LIN {X 0,Y 83.4,Z 651.34,A -85,B 0,C 180,E1 -27838.974,E2 -27838.974} C_VEL
LIN {X 0,Y 87.355,Z 640.881,A -85,B 0,C 180,E1 -27845.629,E2 -27845.629} C_VEL
LIN {X 0,Y 92.332,Z 628.192,A -85,B 0,C 180,E1 -27851.751,E2 -27851.751} C_VEL
LIN {X 0,Y 97.709,Z 614.337,A -85,B 0,C 180,E1 -27856.732,E2 -27856.732} C_VEL
LIN {X 0,Y 102.843,Z 599.666,A -85,B 0,C 180,E1 -27860.677,E2 -27860.677} C_VEL
LIN {X 0,Y 107.389,Z 585.24,A -85,B 0,C 180,E1 -27863.541,E2 -27863.541} C_VEL
LIN {X 0,Y 110.995,Z 571.561,A -85,B 0,C 180,E1 -27865.587,E2 -27865.587} C_VEL
LIN {X 0,Y 111.796,Z 565.957,A -85,B 0,C 180,E1 -27866.44,E2 -27866.44} C_VEL
LIN {X 0,Y 111.242,Z 556.652,A -85,B 0,C 180,E1 -27868.182,E2 -27868.182} C_VEL
LIN {X 0,Y 110.441,Z 547.232,A -85,B 0,C 180,E1 -27869.834,E2 -27869.834} C_VEL
LIN {X 0,Y 110.751,Z 541.433,A -85,B 0,C 180,E1 -27870.482,E2 -27870.482} C_VEL
LIN {X 0,Y 118.536,Z 490.469,A -85,B 0,C 180,E1 -27874.19,E2 -27874.19} C_VEL
LIN {X 0,Y 112.616,Z 471.763,A -85,B 0,C 180,E1 -27879.39,E2 -27879.39} C_VEL
LIN {X 0,Y 109.271,Z 463.872,A -85,B 0,C 180,E1 -27882.247,E2 -27882.247} C_VEL
LIN {X 0,Y 104.426,Z 453.54,A -85,B 0,C 180,E1 -27886.806,E2 -27886.806} C_VEL
LIN {X 0,Y 99.664,Z 444.282,A -85,B 0,C 180,E1 -27891.893,E2 -27891.893} C_VEL
LIN {X 0,Y 95.134,Z 435.831,A -85,B 0,C 180,E1 -27897.713,E2 -27897.713} C_VEL
LIN {X 0,Y 91.912,Z 430.585,A -85,B 0,C 180,E1 -27902.471,E2 -27902.471} C_VEL
LIN {X 0,Y 90.145,Z 427.655,A -85,B 0,C 180,E1 -27905.52,E2 -27905.52} C_VEL
LIN {X 0,Y 87.765,Z 424.651,A -85,B 0,C 180,E1 -27910.178,E2 -27910.178} C_VEL
LIN {X 0,Y 87.158,Z 423.342,A -85,B 0,C 180,E1 -27911.706,E2 -27911.706} C_VEL
LIN {X 0,Y 83.913,Z 420.372,A -85,B 0,C 180,E1 -27920.293,E2 -27920.293} C_VEL
LIN {X 0,Y 83.066,Z 418.058,A -85,B 0,C 180,E1 -27925.028,E2 -27925.028} C_VEL
LIN {X 0,Y 81.987,Z 417.702,A -85,B 0,C 180,E1 -27939.525,E2 -27939.525} C_VEL
LIN {X 0,Y 82.984,Z 418.172,A -85,B 0,C 180,E1 -27946.706,E2 -27946.706} C_VEL
LIN {X 0,Y 84.247,Z 421.149,A -85,B 0,C 180,E1 -27953.039,E2 -27953.039} C_VEL
LIN {X 0,Y 86.921,Z 423.772,A -85,B 0,C 180,E1 -27959.99,E2 -27959.99} C_VEL
LIN {X 0,Y 88.86,Z 427.056,A -85,B 0,C 180,E1 -27964.348,E2 -27964.348} C_VEL
LIN {X 0,Y 90.285,Z 428.713,A -85,B 0,C 180,E1 -27966.89,E2 -27966.89} C_VEL
LIN {X 0,Y 92.73,Z 432.159,A -85,B 0,C 180,E1 -27970.786,E2 -27970.786} C_VEL
LIN {X 0,Y 96.209,Z 437.6,A -85,B 0,C 180,E1 -27975.639,E2 -27975.639} C_VEL
LIN {X 0,Y 99.737,Z 443.153,A -85,B 0,C 180,E1 -27979.836,E2 -27979.836} C_VEL
LIN {X 0,Y 105.389,Z 454.817,A -85,B 0,C 180,E1 -27985.913,E2 -27985.913} C_VEL
LIN {X 0,Y 111.16,Z 468.054,A -85,B 0,C 180,E1 -27991.255,E2 -27991.255} C_VEL
LIN {X 0,Y 116.833,Z 481.707,A -85,B 0,C 180,E1 -27995.829,E2 -27995.829} C_VEL
LIN {X 0,Y 118.524,Z 486.01,A -85,B 0,C 180,E1 -27997.101,E2 -27997.101} C_VEL
LIN {X 0,Y 108.606,Z 548.727,A -85,B 0,C 180,E1 -28001.636,E2 -28001.636} C_VEL
LIN {X 0,Y 105.23,Z 564.977,A -85,B 0,C 180,E1 -28003.441,E2 -28003.441} C_VEL
LIN {X 0,Y 100.84,Z 581.24,A -85,B 0,C 180,E1 -28005.969,E2 -28005.969} C_VEL
LIN {X 0,Y 95.78,Z 596.719,A -85,B 0,C 180,E1 -28009.296,E2 -28009.296} C_VEL
LIN {X 0,Y 90.179,Z 611.69,A -85,B 0,C 180,E1 -28013.687,E2 -28013.687} C_VEL
LIN {X 0,Y 84.987,Z 624.642,A -85,B 0,C 180,E1 -28018.821,E2 -28018.821} C_VEL
LIN {X 0,Y 79.8,Z 637.202,A -85,B 0,C 180,E1 -28025.445,E2 -28025.445} C_VEL
LIN {X 0,Y 75.323,Z 648.898,A -85,B 0,C 180,E1 -28033.686,E2 -28033.686} C_VEL
LIN {X 0,Y 72.406,Z 658.262,A -85,B 0,C 180,E1 -28042.329,E2 -28042.329} C_VEL
LIN {X 0,Y 70.888,Z 665.175,A -85,B 0,C 180,E1 -28050.282,E2 -28050.282} C_VEL
LIN {X 0,Y 70.041,Z 671.752,A -85,B 0,C 180,E1 -28059.438,E2 -28059.438} C_VEL
LIN {X 0,Y 70.296,Z 677.109,A -85,B 0,C 180,E1 -28068.464,E2 -28068.464} C_VEL
LIN {X 0,Y 72.587,Z 682.826,A -85,B 0,C 180,E1 -28079.998,E2 -28079.998} C_VEL
LIN {X 0,Y 77.201,Z 687.278,A -85,B 0,C 180,E1 -28090.489,E2 -28090.489} C_VEL
LIN {X 0,Y 84.118,Z 690.712,A -85,B 0,C 180,E1 -28099.522,E2 -28099.522} C_VEL
LIN {X 0,Y 92.853,Z 693.253,A -85,B 0,C 180,E1 -28107.008,E2 -28107.008} C_VEL
LIN {X 0,Y 104.49,Z 695.039,A -85,B 0,C 180,E1 -28113.751,E2 -28113.751} C_VEL
LIN {X 0,Y 103.442,Z 695.069,A -85,B 0,C 180,E1 -28115.374,E2 -28115.374} C_VEL
LIN {X 0,Y 93.415,Z 694.243,A -85,B 0,C 180,E1 -28121.198,E2 -28121.198} C_VEL
LIN {X 0,Y 84.648,Z 692.545,A -85,B 0,C 180,E1 -28128.37,E2 -28128.37} C_VEL
LIN {X 0,Y 77.842,Z 690.142,A -85,B 0,C 180,E1 -28137.191,E2 -28137.191} C_VEL
LIN {X 0,Y 72.686,Z 685.827,A -85,B 0,C 180,E1 -28150.211,E2 -28150.211} C_VEL
LIN {X 0,Y 71.425,Z 680.817,A -85,B 0,C 180,E1 -28162.373,E2 -28162.373} C_VEL
LIN {X 0,Y 71.518,Z 678.411,A -85,B 0,C 180,E1 -28167.175,E2 -28167.175} C_VEL
LIN {X 0,Y 71.275,Z 673.088,A -85,B 0,C 180,E1 -28175.65,E2 -28175.65} C_VEL
LIN {X 0,Y 72.103,Z 665.419,A -85,B 0,C 180,E1 -28185.539,E2 -28185.539} C_VEL
LIN {X 0,Y 74.517,Z 655.967,A -85,B 0,C 180,E1 -28195.104,E2 -28195.104} C_VEL
LIN {X 0,Y 78.723,Z 644.592,A -85,B 0,C 180,E1 -28203.906,E2 -28203.906} C_VEL
LIN {X 0,Y 83.249,Z 633.196,A -85,B 0,C 180,E1 -28210.556,E2 -28210.556} C_VEL
LIN {X 0,Y 88.734,Z 620.083,A -85,B 0,C 180,E1 -28216.27,E2 -28216.27} C_VEL
LIN {X 0,Y 93.537,Z 607.632,A -85,B 0,C 180,E1 -28220.356,E2 -28220.356} C_VEL
LIN {X 0,Y 98.821,Z 592.668,A -85,B 0,C 180,E1 -28223.984,E2 -28223.984} C_VEL
LIN {X 0,Y 103.223,Z 577.827,A -85,B 0,C 180,E1 -28226.649,E2 -28226.649} C_VEL
LIN {X 0,Y 106.858,Z 562.938,A -85,B 0,C 180,E1 -28228.602,E2 -28228.602} C_VEL
LIN {X 0,Y 109.639,Z 548.688,A -85,B 0,C 180,E1 -28229.913,E2 -28229.913} C_VEL
LIN {X 0,Y 110.751,Z 541.433,A -85,B 0,C 180,E1 -28230.482,E2 -28230.482} C_VEL
LIN {X 0,Y 111.09,Z 535.664,A -85,B 0,C 180,E1 -28231.12,E2 -28231.12} C_VEL
LIN {X 0,Y 109.501,Z 516.872,A -85,B 0,C 180,E1 -28234.326,E2 -28234.326} C_VEL
LIN {X 0,Y 109.908,Z 511.103,A -85,B 0,C 180,E1 -28234.962,E2 -28234.962} C_VEL
LIN {X 0,Y 112.849,Z 492.252,A -85,B 0,C 180,E1 -28236.331,E2 -28236.331} C_VEL
LIN {X 0,Y 107.793,Z 475.639,A -85,B 0,C 180,E1 -28241.188,E2 -28241.188} C_VEL
LIN {X 0,Y 104.92,Z 468.523,A -85,B 0,C 180,E1 -28243.921,E2 -28243.921} C_VEL
LIN {X 0,Y 100.246,Z 458.053,A -85,B 0,C 180,E1 -28248.824,E2 -28248.824} C_VEL
LIN {X 0,Y 95.193,Z 447.833,A -85,B 0,C 180,E1 -28254.835,E2 -28254.835} C_VEL
LIN {X 0,Y 91.737,Z 441.143,A -85,B 0,C 180,E1 -28259.869,E2 -28259.869} C_VEL
LIN {X 0,Y 89.106,Z 436.502,A -85,B 0,C 180,E1 -28264.187,E2 -28264.187} C_VEL
LIN {X 0,Y 87.569,Z 433.904,A -85,B 0,C 180,E1 -28267.147,E2 -28267.147} C_VEL
LIN {X 0,Y 85.254,Z 430.535,A -85,B 0,C 180,E1 -28272.22,E2 -28272.22} C_VEL
LIN {X 0,Y 84.709,Z 429.774,A -85,B 0,C 180,E1 -28273.543,E2 -28273.543} C_VEL
LIN {X 0,Y 82.042,Z 426.845,A -85,B 0,C 180,E1 -28281.915,E2 -28281.915} C_VEL
LIN {X 0,Y 81.443,Z 425.088,A -85,B 0,C 180,E1 -28285.562,E2 -28285.562} C_VEL
LIN {X 0,Y 80.477,Z 424.626,A -85,B 0,C 180,E1 -28298.203,E2 -28298.203} C_VEL
LIN {X 0,Y 81.333,Z 425.135,A -85,B 0,C 180,E1 -28305.96,E2 -28305.96} C_VEL
LIN {X 0,Y 83.041,Z 428.687,A -85,B 0,C 180,E1 -28314.159,E2 -28314.159} C_VEL
LIN {X 0,Y 84.78,Z 430.442,A -85,B 0,C 180,E1 -28318.804,E2 -28318.804} C_VEL
LIN {X 0,Y 86.896,Z 433.84,A -85,B 0,C 180,E1 -28323.684,E2 -28323.684} C_VEL
LIN {X 0,Y 87.932,Z 435.321,A -85,B 0,C 180,E1 -28325.758,E2 -28325.758} C_VEL
LIN {X 0,Y 90.71,Z 439.474,A -85,B 0,C 180,E1 -28330.503,E2 -28330.503} C_VEL
LIN {X 0,Y 93.875,Z 444.671,A -85,B 0,C 180,E1 -28335.078,E2 -28335.078} C_VEL
LIN {X 0,Y 96.373,Z 448.911,A -85,B 0,C 180,E1 -28338.317,E2 -28338.317} C_VEL
LIN {X 0,Y 101.476,Z 460.012,A -85,B 0,C 180,E1 -28344.265,E2 -28344.265} C_VEL
LIN {X 0,Y 106.79,Z 472.868,A -85,B 0,C 180,E1 -28349.725,E2 -28349.725} C_VEL
LIN {X 0,Y 112.767,Z 487.766,A -85,B 0,C 180,E1 -28354.863,E2 -28354.863} C_VEL
LIN {X 0,Y 104.427,Z 539.915,A -85,B 0,C 180,E1 -28358.697,E2 -28358.697} C_VEL
LIN {X 0,Y 101.113,Z 557.125,A -85,B 0,C 180,E1 -28360.273,E2 -28360.273} C_VEL
LIN {X 0,Y 97.417,Z 572.043,A -85,B 0,C 180,E1 -28362.273,E2 -28362.273} C_VEL
LIN {X 0,Y 92.422,Z 588.129,A -85,B 0,C 180,E1 -28365.244,E2 -28365.244} C_VEL
LIN {X 0,Y 86.759,Z 603.763,A -85,B 0,C 180,E1 -28369.273,E2 -28369.273} C_VEL
LIN {X 0,Y 80.958,Z 617.943,A -85,B 0,C 180,E1 -28374.287,E2 -28374.287} C_VEL
LIN {X 0,Y 75.457,Z 630.788,A -85,B 0,C 180,E1 -28380.507,E2 -28380.507} C_VEL
LIN {X 0,Y 70.887,Z 641.562,A -85,B 0,C 180,E1 -28387.517,E2 -28387.517} C_VEL
LIN {X 0,Y 67.145,Z 651.543,A -85,B 0,C 180,E1 -28396.049,E2 -28396.049} C_VEL
LIN {X 0,Y 64.435,Z 661.363,A -85,B 0,C 180,E1 -28406.949,E2 -28406.949} C_VEL
LIN {X 0,Y 63.243,Z 668.627,A -85,B 0,C 180,E1 -28417.109,E2 -28417.109} C_VEL
LIN {X 0,Y 63.267,Z 674.398,A -85,B 0,C 180,E1 -28427.162,E2 -28427.162} C_VEL
LIN {X 0,Y 65.417,Z 680.637,A -85,B 0,C 180,E1 -28439.998,E2 -28439.998} C_VEL
LIN {X 0,Y 70.149,Z 685.571,A -85,B 0,C 180,E1 -28451.557,E2 -28451.557} C_VEL
LIN {X 0,Y 77.355,Z 689.428,A -85,B 0,C 180,E1 -28461.309,E2 -28461.309} C_VEL
LIN {X 0,Y 86.428,Z 692.389,A -85,B 0,C 180,E1 -28469.201,E2 -28469.201} C_VEL
LIN {X 0,Y 91.847,Z 693.586,A -85,B 0,C 180,E1 -28472.668,E2 -28472.668} C_VEL
LIN {X 0,Y 94.095,Z 694.045,A -85,B 0,C 180,E1 -28474.745,E2 -28474.745} C_VEL
LIN {X 0,Y 79.518,Z 691.492,A -85,B 0,C 180,E1 -28484.994,E2 -28484.994} C_VEL
LIN {X 0,Y 69.224,Z 687.122,A -85,B 0,C 180,E1 -28499.485,E2 -28499.485} C_VEL
LIN {X 0,Y 65.545,Z 683.066,A -85,B 0,C 180,E1 -28511.226,E2 -28511.226} C_VEL
LIN {X 0,Y 64.721,Z 677.982,A -85,B 0,C 180,E1 -28523.757,E2 -28523.757} C_VEL
LIN {X 0,Y 64.541,Z 674.68,A -85,B 0,C 180,E1 -28529.991,E2 -28529.991} C_VEL
LIN {X 0,Y 64.449,Z 669.034,A -85,B 0,C 180,E1 -28538.816,E2 -28538.816} C_VEL
LIN {X 0,Y 65.361,Z 662.721,A -85,B 0,C 180,E1 -28547.19,E2 -28547.19} C_VEL
LIN {X 0,Y 68.239,Z 652.923,A -85,B 0,C 180,E1 -28557.6,E2 -28557.6} C_VEL
LIN {X 0,Y 72.206,Z 642.852,A -85,B 0,C 180,E1 -28565.721,E2 -28565.721} C_VEL
LIN {X 0,Y 77.472,Z 630.305,A -85,B 0,C 180,E1 -28573.246,E2 -28573.246} C_VEL
LIN {X 0,Y 82.941,Z 617.719,A -85,B 0,C 180,E1 -28578.754,E2 -28578.754} C_VEL
LIN {X 0,Y 88.624,Z 603.293,A -85,B 0,C 180,E1 -28583.398,E2 -28583.398} C_VEL
LIN {X 0,Y 94.231,Z 587.487,A -85,B 0,C 180,E1 -28587.028,E2 -28587.028} C_VEL
LIN {X 0,Y 99.038,Z 570.951,A -85,B 0,C 180,E1 -28589.755,E2 -28589.755} C_VEL
LIN {X 0,Y 102.85,Z 554.608,A -85,B 0,C 180,E1 -28591.605,E2 -28591.605} C_VEL
LIN {X 0,Y 109.908,Z 511.103,A -85,B 0,C 180,E1 -28594.962,E2 -28594.962} C_VEL
LIN {X 0,Y 110.223,Z 507.254,A -85,B 0,C 180,E1 -28595.373,E2 -28595.373} C_VEL
LIN {X 0,Y 109.773,Z 501.658,A -85,B 0,C 180,E1 -28596.38,E2 -28596.38} C_VEL
LIN {X 0,Y 108.55,Z 496.379,A -85,B 0,C 180,E1 -28597.708,E2 -28597.708} C_VEL
LIN {X 0,Y 104.028,Z 482.75,A -85,B 0,C 180,E1 -28602.073,E2 -28602.073} C_VEL
LIN {X 0,Y 101.897,Z 476.229,A -85,B 0,C 180,E1 -28604.416,E2 -28604.416} C_VEL
LIN {X 0,Y 97.693,Z 466.124,A -85,B 0,C 180,E1 -28609.06,E2 -28609.06} C_VEL
LIN {X 0,Y 93.087,Z 455.985,A -85,B 0,C 180,E1 -28614.877,E2 -28614.877} C_VEL
LIN {X 0,Y 88.893,Z 447.211,A -85,B 0,C 180,E1 -28621.353,E2 -28621.353} C_VEL
LIN {X 0,Y 85.396,Z 440.486,A -85,B 0,C 180,E1 -28628.172,E2 -28628.172} C_VEL
LIN {X 0,Y 82.991,Z 436.835,A -85,B 0,C 180,E1 -28633.829,E2 -28633.829} C_VEL
LIN {X 0,Y 80.039,Z 432.914,A -85,B 0,C 180,E1 -28644.512,E2 -28644.512} C_VEL
LIN {X 0,Y 79.66,Z 431.821,A -85,B 0,C 180,E1 -28647.249,E2 -28647.249} C_VEL
LIN {X 0,Y 79.032,Z 431.568,A -85,B 0,C 180,E1 -28658.499,E2 -28658.499} C_VEL
LIN {X 0,Y 79.693,Z 432.069,A -85,B 0,C 180,E1 -28665.141,E2 -28665.141} C_VEL
LIN {X 0,Y 81.687,Z 435.942,A -85,B 0,C 180,E1 -28674.737,E2 -28674.737} C_VEL
LIN {X 0,Y 82.616,Z 436.923,A -85,B 0,C 180,E1 -28677.368,E2 -28677.368} C_VEL
LIN {X 0,Y 84.684,Z 440.337,A -85,B 0,C 180,E1 -28682.492,E2 -28682.492} C_VEL
LIN {X 0,Y 87.851,Z 445.4,A -85,B 0,C 180,E1 -28688.793,E2 -28688.793} C_VEL
LIN {X 0,Y 91.961,Z 452.355,A -85,B 0,C 180,E1 -28695.059,E2 -28695.059} C_VEL
LIN {X 0,Y 95.16,Z 459.605,A -85,B 0,C 180,E1 -28699.602,E2 -28699.602} C_VEL
LIN {X 0,Y 98.909,Z 468.618,A -85,B 0,C 180,E1 -28704.153,E2 -28704.153} C_VEL
LIN {X 0,Y 103.142,Z 479.356,A -85,B 0,C 180,E1 -28708.74,E2 -28708.74} C_VEL
LIN {X 0,Y 107.174,Z 489.956,A -85,B 0,C 180,E1 -28712.58,E2 -28712.58} C_VEL
LIN {X 0,Y 97.537,Z 546.504,A -85,B 0,C 180,E1 -28716.792,E2 -28716.792} C_VEL
LIN {X 0,Y 93.909,Z 563.2,A -85,B 0,C 180,E1 -28718.615,E2 -28718.615} C_VEL
LIN {X 0,Y 89.493,Z 578.67,A -85,B 0,C 180,E1 -28720.988,E2 -28720.988} C_VEL
LIN {X 0,Y 84.193,Z 594.018,A -85,B 0,C 180,E1 -28724.27,E2 -28724.27} C_VEL
LIN {X 0,Y 78.687,Z 607.907,A -85,B 0,C 180,E1 -28728.375,E2 -28728.375} C_VEL
LIN {X 0,Y 72.79,Z 621.401,A -85,B 0,C 180,E1 -28733.928,E2 -28733.928} C_VEL
LIN {X 0,Y 67.266,Z 633.472,A -85,B 0,C 180,E1 -28740.755,E2 -28740.755} C_VEL
LIN {X 0,Y 62.856,Z 643.63,A -85,B 0,C 180,E1 -28748.491,E2 -28748.491} C_VEL
LIN {X 0,Y 58.974,Z 654.059,A -85,B 0,C 180,E1 -28759.045,E2 -28759.045} C_VEL
LIN {X 0,Y 57.067,Z 662.089,A -85,B 0,C 180,E1 -28769.57,E2 -28769.57} C_VEL
LIN {X 0,Y 56.252,Z 668.459,A -85,B 0,C 180,E1 -28779.903,E2 -28779.903} C_VEL
LIN {X 0,Y 56.928,Z 675.031,A -85,B 0,C 180,E1 -28792.906,E2 -28792.906} C_VEL
LIN {X 0,Y 60.395,Z 681.051,A -85,B 0,C 180,E1 -28806.681,E2 -28806.681} C_VEL
LIN {X 0,Y 66.738,Z 685.963,A -85,B 0,C 180,E1 -28818.575,E2 -28818.575} C_VEL
LIN {X 0,Y 80.183,Z 691.258,A -85,B 0,C 180,E1 -28831.727,E2 -28831.727} C_VEL
LIN {X 0,Y 83.422,Z 692.126,A -85,B 0,C 180,E1 -28833.87,E2 -28833.87} C_VEL
LIN {X 0,Y 82.706,Z 692.041,A -85,B 0,C 180,E1 -28835.271,E2 -28835.271} C_VEL
LIN {X 0,Y 70.348,Z 688.871,A -85,B 0,C 180,E1 -28845.616,E2 -28845.616} C_VEL
LIN {X 0,Y 61.987,Z 684.558,A -85,B 0,C 180,E1 -28859.312,E2 -28859.312} C_VEL
LIN {X 0,Y 58.146,Z 678.749,A -85,B 0,C 180,E1 -28876.001,E2 -28876.001} C_VEL
LIN {X 0,Y 57.98,Z 675.904,A -85,B 0,C 180,E1 -28883.027,E2 -28883.027} C_VEL
LIN {X 0,Y 57.654,Z 672.44,A -85,B 0,C 180,E1 -28889.99,E2 -28889.99} C_VEL
LIN {X 0,Y 57.853,Z 664.848,A -85,B 0,C 180,E1 -28902.383,E2 -28902.383} C_VEL
LIN {X 0,Y 59.921,Z 655.642,A -85,B 0,C 180,E1 -28914.226,E2 -28914.226} C_VEL
LIN {X 0,Y 63.499,Z 646.207,A -85,B 0,C 180,E1 -28923.589,E2 -28923.589} C_VEL
LIN {X 0,Y 68.404,Z 635.031,A -85,B 0,C 180,E1 -28931.887,E2 -28931.887} C_VEL
LIN {X 0,Y 74.016,Z 622.74,A -85,B 0,C 180,E1 -28938.507,E2 -28938.507} C_VEL
LIN {X 0,Y 79.672,Z 609.635,A -85,B 0,C 180,E1 -28943.59,E2 -28943.59} C_VEL
LIN {X 0,Y 85.281,Z 595.268,A -85,B 0,C 180,E1 -28947.625,E2 -28947.625} C_VEL
LIN {X 0,Y 90.263,Z 580.691,A -85,B 0,C 180,E1 -28950.569,E2 -28950.569} C_VEL
LIN {X 0,Y 94.704,Z 564.576,A -85,B 0,C 180,E1 -28952.924,E2 -28952.924} C_VEL
LIN {X 0,Y 98.01,Z 549.43,A -85,B 0,C 180,E1 -28954.432,E2 -28954.432} C_VEL
LIN {X 0,Y 107.266,Z 493.905,A -85,B 0,C 180,E1 -28958.669,E2 -28958.669} C_VEL
LIN {X 0,Y 104.028,Z 482.75,A -85,B 0,C 180,E1 -28962.073,E2 -28962.073} C_VEL
LIN {X 0,Y 102.842,Z 479.687,A -85,B 0,C 180,E1 -28963.257,E2 -28963.257} C_VEL
LIN {X 0,Y 101.281,Z 477.066,A -85,B 0,C 180,E1 -28964.65,E2 -28964.65} C_VEL
LIN {X 0,Y 97.595,Z 472.757,A -85,B 0,C 180,E1 -28967.863,E2 -28967.863} C_VEL
LIN {X 0,Y 92.154,Z 466.593,A -85,B 0,C 180,E1 -28973.301,E2 -28973.301} C_VEL
LIN {X 0,Y 90.821,Z 464.06,A -85,B 0,C 180,E1 -28975.089,E2 -28975.089} C_VEL
LIN {X 0,Y 87.082,Z 455.522,A -85,B 0,C 180,E1 -28981.123,E2 -28981.123} C_VEL
LIN {X 0,Y 84.081,Z 449.056,A -85,B 0,C 180,E1 -28987.141,E2 -28987.141} C_VEL
LIN {X 0,Y 82.634,Z 446.346,A -85,B 0,C 180,E1 -28990.546,E2 -28990.546} C_VEL
LIN {X 0,Y 80.518,Z 442.925,A -85,B 0,C 180,E1 -28996.261,E2 -28996.261} C_VEL
LIN {X 0,Y 78.408,Z 439.849,A -85,B 0,C 180,E1 -29005.056,E2 -29005.056} C_VEL
LIN {X 0,Y 78.132,Z 438.722,A -85,B 0,C 180,E1 -29007.544,E2 -29007.544} C_VEL
LIN {X 0,Y 77.592,Z 438.548,A -85,B 0,C 180,E1 -29019.35,E2 -29019.35} C_VEL
LIN {X 0,Y 78.054,Z 438.9,A -85,B 0,C 180,E1 -29024.166,E2 -29024.166} C_VEL
LIN {X 0,Y 80,Z 442.817,A -85,B 0,C 180,E1 -29034.273,E2 -29034.273} C_VEL
LIN {X 0,Y 80.584,Z 443.656,A -85,B 0,C 180,E1 -29036.173,E2 -29036.173} C_VEL
LIN {X 0,Y 83.15,Z 448.015,A -85,B 0,C 180,E1 -29042.862,E2 -29042.862} C_VEL
LIN {X 0,Y 85.387,Z 452.007,A -85,B 0,C 180,E1 -29047.626,E2 -29047.626} C_VEL
LIN {X 0,Y 89.135,Z 458.751,A -85,B 0,C 180,E1 -29053.85,E2 -29053.85} C_VEL
LIN {X 0,Y 93.266,Z 469.238,A -85,B 0,C 180,E1 -29060.117,E2 -29060.117} C_VEL
LIN {X 0,Y 97.709,Z 481.044,A -85,B 0,C 180,E1 -29065.657,E2 -29065.657} C_VEL
LIN {X 0,Y 101.664,Z 491.965,A -85,B 0,C 180,E1 -29070.006,E2 -29070.006} C_VEL
LIN {X 0,Y 92.249,Z 545.502,A -85,B 0,C 180,E1 -29073.99,E2 -29073.99} C_VEL
LIN {X 0,Y 88.314,Z 563.044,A -85,B 0,C 180,E1 -29075.865,E2 -29075.865} C_VEL
LIN {X 0,Y 83.737,Z 578.397,A -85,B 0,C 180,E1 -29078.236,E2 -29078.236} C_VEL
LIN {X 0,Y 78.051,Z 594.121,A -85,B 0,C 180,E1 -29081.692,E2 -29081.692} C_VEL
LIN {X 0,Y 72.056,Z 608.35,A -85,B 0,C 180,E1 -29086.115,E2 -29086.115} C_VEL
LIN {X 0,Y 65.548,Z 622.429,A -85,B 0,C 180,E1 -29092.362,E2 -29092.362} C_VEL
LIN {X 0,Y 60.129,Z 633.728,A -85,B 0,C 180,E1 -29099.376,E2 -29099.376} C_VEL
LIN {X 0,Y 55.616,Z 643.71,A -85,B 0,C 180,E1 -29107.83,E2 -29107.83} C_VEL
LIN {X 0,Y 51.683,Z 654.011,A -85,B 0,C 180,E1 -29119.762,E2 -29119.762} C_VEL
LIN {X 0,Y 49.98,Z 661.315,A -85,B 0,C 180,E1 -29130.728,E2 -29130.728} C_VEL
LIN {X 0,Y 49.357,Z 668.196,A -85,B 0,C 180,E1 -29143.452,E2 -29143.452} C_VEL
LIN {X 0,Y 50.449,Z 673.878,A -85,B 0,C 180,E1 -29156.004,E2 -29156.004} C_VEL
LIN {X 0,Y 54.731,Z 680.068,A -85,B 0,C 180,E1 -29171.103,E2 -29171.103} C_VEL
LIN {X 0,Y 64.175,Z 686.139,A -85,B 0,C 180,E1 -29185.978,E2 -29185.978} C_VEL
LIN {X 0,Y 72.799,Z 689.489,A -85,B 0,C 180,E1 -29193.716,E2 -29193.716} C_VEL
LIN {X 0,Y 70.312,Z 688.905,A -85,B 0,C 180,E1 -29196.891,E2 -29196.891} C_VEL
LIN {X 0,Y 57.716,Z 683.811,A -85,B 0,C 180,E1 -29212.482,E2 -29212.482} C_VEL
LIN {X 0,Y 52.746,Z 679.298,A -85,B 0,C 180,E1 -29226.427,E2 -29226.427} C_VEL
LIN {X 0,Y 51.285,Z 673.685,A -85,B 0,C 180,E1 -29242.112,E2 -29242.112} C_VEL
LIN {X 0,Y 50.807,Z 670.005,A -85,B 0,C 180,E1 -29249.988,E2 -29249.988} C_VEL
LIN {X 0,Y 51.013,Z 662.528,A -85,B 0,C 180,E1 -29263.361,E2 -29263.361} C_VEL
LIN {X 0,Y 53.66,Z 652.473,A -85,B 0,C 180,E1 -29277.271,E2 -29277.271} C_VEL
LIN {X 0,Y 57.809,Z 642.526,A -85,B 0,C 180,E1 -29287.421,E2 -29287.421} C_VEL
LIN {X 0,Y 62.827,Z 631.726,A -85,B 0,C 180,E1 -29295.476,E2 -29295.476} C_VEL
LIN {X 0,Y 69.339,Z 618.186,A -85,B 0,C 180,E1 -29302.62,E2 -29302.62} C_VEL
LIN {X 0,Y 75.063,Z 605.299,A -85,B 0,C 180,E1 -29307.405,E2 -29307.405} C_VEL
LIN {X 0,Y 81.086,Z 590.294,A -85,B 0,C 180,E1 -29311.334,E2 -29311.334} C_VEL
LIN {X 0,Y 85.955,Z 575.61,A -85,B 0,C 180,E1 -29314.062,E2 -29314.062} C_VEL
LIN {X 0,Y 90.083,Z 560.259,A -85,B 0,C 180,E1 -29316.083,E2 -29316.083} C_VEL
LIN {X 0,Y 93.144,Z 545.59,A -85,B 0,C 180,E1 -29317.428,E2 -29317.428} C_VEL
LIN {X 0,Y 101.713,Z 496.179,A -85,B 0,C 180,E1 -29321.142,E2 -29321.142} C_VEL
LIN {X 0,Y 101.348,Z 493.99,A -85,B 0,C 180,E1 -29321.71,E2 -29321.71} C_VEL
LIN {X 0,Y 97.831,Z 481.263,A -85,B 0,C 180,E1 -29326.13,E2 -29326.13} C_VEL
LIN {X 0,Y 93.378,Z 470.18,A -85,B 0,C 180,E1 -29331.479,E2 -29331.479} C_VEL
LIN {X 0,Y 90.821,Z 464.06,A -85,B 0,C 180,E1 -29335.089,E2 -29335.089} C_VEL
LIN {X 0,Y 88.874,Z 460.602,A -85,B 0,C 180,E1 -29337.875,E2 -29337.875} C_VEL
LIN {X 0,Y 86.588,Z 458.063,A -85,B 0,C 180,E1 -29341.051,E2 -29341.051} C_VEL
LIN {X 0,Y 79.781,Z 451.905,A -85,B 0,C 180,E1 -29353.49,E2 -29353.49} C_VEL
LIN {X 0,Y 78.564,Z 449.575,A -85,B 0,C 180,E1 -29357.485,E2 -29357.485} C_VEL
LIN {X 0,Y 76.714,Z 446.557,A -85,B 0,C 180,E1 -29366.188,E2 -29366.188} C_VEL
LIN {X 0,Y 76.418,Z 445.62,A -85,B 0,C 180,E1 -29369.06,E2 -29369.06} C_VEL
LIN {X 0,Y 76.389,Z 445.619,A -85,B 0,C 180,E1 -29382.619,E2 -29382.619} C_VEL
LIN {X 0,Y 78.604,Z 450.266,A -85,B 0,C 180,E1 -29394.901,E2 -29394.901} C_VEL
LIN {X 0,Y 80.77,Z 454.415,A -85,B 0,C 180,E1 -29401.356,E2 -29401.356} C_VEL
LIN {X 0,Y 82.703,Z 458.009,A -85,B 0,C 180,E1 -29405.799,E2 -29405.799} C_VEL
LIN {X 0,Y 85.89,Z 464.462,A -85,B 0,C 180,E1 -29411.92,E2 -29411.92} C_VEL
LIN {X 0,Y 89.304,Z 473.658,A -85,B 0,C 180,E1 -29417.672,E2 -29417.672} C_VEL
LIN {X 0,Y 93.399,Z 485.494,A -85,B 0,C 180,E1 -29423.587,E2 -29423.587} C_VEL
LIN {X 0,Y 96.42,Z 494.278,A -85,B 0,C 180,E1 -29427.254,E2 -29427.254} C_VEL
LIN {X 0,Y 86.525,Z 547.166,A -85,B 0,C 180,E1 -29431.132,E2 -29431.132} C_VEL
LIN {X 0,Y 82.517,Z 563.903,A -85,B 0,C 180,E1 -29432.976,E2 -29432.976} C_VEL
LIN {X 0,Y 77.657,Z 579.397,A -85,B 0,C 180,E1 -29435.417,E2 -29435.417} C_VEL
LIN {X 0,Y 72,Z 594.28,A -85,B 0,C 180,E1 -29438.759,E2 -29438.759} C_VEL
LIN {X 0,Y 65.802,Z 608.275,A -85,B 0,C 180,E1 -29443.209,E2 -29443.209} C_VEL
LIN {X 0,Y 58.73,Z 622.743,A -85,B 0,C 180,E1 -29449.989,E2 -29449.989} C_VEL
LIN {X 0,Y 52.247,Z 635.505,A -85,B 0,C 180,E1 -29459.028,E2 -29459.028} C_VEL
LIN {X 0,Y 46.798,Z 647.202,A -85,B 0,C 180,E1 -29471.329,E2 -29471.329} C_VEL
LIN {X 0,Y 43.525,Z 657.56,A -85,B 0,C 180,E1 -29486.851,E2 -29486.851} C_VEL
LIN {X 0,Y 42.552,Z 664.662,A -85,B 0,C 180,E1 -29500.709,E2 -29500.709} C_VEL
LIN {X 0,Y 43.424,Z 670.764,A -85,B 0,C 180,E1 -29515.356,E2 -29515.356} C_VEL
LIN {X 0,Y 47.847,Z 677.513,A -85,B 0,C 180,E1 -29532.726,E2 -29532.726} C_VEL
LIN {X 0,Y 57.857,Z 684.11,A -85,B 0,C 180,E1 -29549.068,E2 -29549.068} C_VEL
LIN {X 0,Y 62.899,Z 686.348,A -85,B 0,C 180,E1 -29553.962,E2 -29553.962} C_VEL
LIN {X 0,Y 61.177,Z 685.774,A -85,B 0,C 180,E1 -29556.456,E2 -29556.456} C_VEL
LIN {X 0,Y 50.645,Z 680.884,A -85,B 0,C 180,E1 -29571.343,E2 -29571.343} C_VEL
LIN {X 0,Y 45.143,Z 674.468,A -85,B 0,C 180,E1 -29591.845,E2 -29591.845} C_VEL
LIN {X 0,Y 44.618,Z 671.407,A -85,B 0,C 180,E1 -29600.924,E2 -29600.924} C_VEL
LIN {X 0,Y 43.869,Z 666.398,A -85,B 0,C 180,E1 -29612.282,E2 -29612.282} C_VEL
LIN {X 0,Y 44.354,Z 659.522,A -85,B 0,C 180,E1 -29625.413,E2 -29625.413} C_VEL
LIN {X 0,Y 46.981,Z 650.541,A -85,B 0,C 180,E1 -29639.074,E2 -29639.074} C_VEL
LIN {X 0,Y 51.542,Z 640.454,A -85,B 0,C 180,E1 -29650.352,E2 -29650.352} C_VEL
LIN {X 0,Y 57.024,Z 629.409,A -85,B 0,C 180,E1 -29658.998,E2 -29658.998} C_VEL
LIN {X 0,Y 63.747,Z 616.156,A -85,B 0,C 180,E1 -29666.028,E2 -29666.028} C_VEL
LIN {X 0,Y 70.176,Z 602.047,A -85,B 0,C 180,E1 -29671.18,E2 -29671.18} C_VEL
LIN {X 0,Y 75.819,Z 588.295,A -85,B 0,C 180,E1 -29674.638,E2 -29674.638} C_VEL
LIN {X 0,Y 80.904,Z 573.344,A -85,B 0,C 180,E1 -29677.345,E2 -29677.345} C_VEL
LIN {X 0,Y 85.227,Z 557.738,A -85,B 0,C 180,E1 -29679.276,E2 -29679.276} C_VEL
LIN {X 0,Y 89.174,Z 537.898,A -85,B 0,C 180,E1 -29681.017,E2 -29681.017} C_VEL
LIN {X 0,Y 96.512,Z 497.355,A -85,B 0,C 180,E1 -29684.007,E2 -29684.007} C_VEL
LIN {X 0,Y 93.38,Z 485.367,A -85,B 0,C 180,E1 -29688.351,E2 -29688.351} C_VEL
LIN {X 0,Y 89.104,Z 473.811,A -85,B 0,C 180,E1 -29694.358,E2 -29694.358} C_VEL
LIN {X 0,Y 85.116,Z 463.828,A -85,B 0,C 180,E1 -29701.06,E2 -29701.06} C_VEL
LIN {X 0,Y 82.614,Z 457.835,A -85,B 0,C 180,E1 -29706.277,E2 -29706.277} C_VEL
LIN {X 0,Y 80.591,Z 453.077,A -85,B 0,C 180,E1 -29711.432,E2 -29711.432} C_VEL
LIN {X 0,Y 79.781,Z 451.905,A -85,B 0,C 180,E1 -29713.49,E2 -29713.49} C_VEL
LIN {X 0,Y 78.346,Z 450.533,A -85,B 0,C 180,E1 -29717.524,E2 -29717.524} C_VEL
LIN {X 0,Y 76.57,Z 450.515,A -85,B 0,C 180,E1 -29723.259,E2 -29723.259} C_VEL
LIN {X 0,Y 74.614,Z 452.263,A -85,B 0,C 180,E1 -29733.913,E2 -29733.913} C_VEL
LIN {X 0,Y 74.521,Z 452.459,A -85,B 0,C 180,E1 -29737.048,E2 -29737.048} C_VEL
LIN {X 0,Y 74.865,Z 452.655,A -85,B 0,C 180,E1 -29742.423,E2 -29742.423} C_VEL
LIN {X 0,Y 76.641,Z 456.833,A -85,B 0,C 180,E1 -29753.467,E2 -29753.467} C_VEL
LIN {X 0,Y 78.388,Z 460.633,A -85,B 0,C 180,E1 -29759.575,E2 -29759.575} C_VEL
LIN {X 0,Y 80.671,Z 465.179,A -85,B 0,C 180,E1 -29765.238,E2 -29765.238} C_VEL
LIN {X 0,Y 82.705,Z 470.007,A -85,B 0,C 180,E1 -29769.736,E2 -29769.736} C_VEL
LIN {X 0,Y 85.73,Z 479.029,A -85,B 0,C 180,E1 -29775.584,E2 -29775.584} C_VEL
LIN {X 0,Y 89.168,Z 489.822,A -85,B 0,C 180,E1 -29781.254,E2 -29781.254} C_VEL
LIN {X 0,Y 91.215,Z 496.211,A -85,B 0,C 180,E1 -29784.17,E2 -29784.17} C_VEL
LIN {X 0,Y 81.547,Z 546.327,A -85,B 0,C 180,E1 -29787.732,E2 -29787.732} C_VEL
LIN {X 0,Y 77.313,Z 563.476,A -85,B 0,C 180,E1 -29789.521,E2 -29789.521} C_VEL
LIN {X 0,Y 71.957,Z 579.893,A -85,B 0,C 180,E1 -29792.032,E2 -29792.032} C_VEL
LIN {X 0,Y 65.687,Z 595.492,A -85,B 0,C 180,E1 -29795.587,E2 -29795.587} C_VEL
LIN {X 0,Y 58.95,Z 609.679,A -85,B 0,C 180,E1 -29800.392,E2 -29800.392} C_VEL
LIN {X 0,Y 51.609,Z 623.646,A -85,B 0,C 180,E1 -29807.584,E2 -29807.584} C_VEL
LIN {X 0,Y 44.39,Z 636.948,A -85,B 0,C 180,E1 -29818.372,E2 -29818.372} C_VEL
LIN {X 0,Y 39.504,Z 647.032,A -85,B 0,C 180,E1 -29830.874,E2 -29830.874} C_VEL
LIN {X 0,Y 36.468,Z 656.676,A -85,B 0,C 180,E1 -29847.993,E2 -29847.993} C_VEL
LIN {X 0,Y 35.796,Z 663.061,A -85,B 0,C 180,E1 -29862.875,E2 -29862.875} C_VEL
LIN {X 0,Y 37.202,Z 669.412,A -85,B 0,C 180,E1 -29879.997,E2 -29879.997} C_VEL
LIN {X 0,Y 42.851,Z 676.206,A -85,B 0,C 180,E1 -29899.146,E2 -29899.146} C_VEL
LIN {X 0,Y 52.769,Z 682.298,A -85,B 0,C 180,E1 -29913.887,E2 -29913.887} C_VEL
LIN {X 0,Y 52.188,Z 682.106,A -85,B 0,C 180,E1 -29916.08,E2 -29916.08} C_VEL
LIN {X 0,Y 42.063,Z 676.327,A -85,B 0,C 180,E1 -29934.194,E2 -29934.194} C_VEL
LIN {X 0,Y 38.305,Z 670.551,A -85,B 0,C 180,E1 -29954.009,E2 -29954.009} C_VEL
LIN {X 0,Y 38.021,Z 668.84,A -85,B 0,C 180,E1 -29959.332,E2 -29959.332} C_VEL
LIN {X 0,Y 37.038,Z 663.61,A -85,B 0,C 180,E1 -29972.703,E2 -29972.703} C_VEL
LIN {X 0,Y 37.841,Z 655.839,A -85,B 0,C 180,E1 -29989.24,E2 -29989.24} C_VEL
LIN {X 0,Y 41.083,Z 646.957,A -85,B 0,C 180,E1 -30003.759,E2 -30003.759} C_VEL
LIN {X 0,Y 46.51,Z 636.308,A -85,B 0,C 180,E1 -30015.851,E2 -30015.851} C_VEL
LIN {X 0,Y 53.386,Z 623.535,A -85,B 0,C 180,E1 -30025.343,E2 -30025.343} C_VEL
LIN {X 0,Y 60.66,Z 609.586,A -85,B 0,C 180,E1 -30031.925,E2 -30031.925} C_VEL
LIN {X 0,Y 67.121,Z 595.429,A -85,B 0,C 180,E1 -30036.35,E2 -30036.35} C_VEL
LIN {X 0,Y 73.119,Z 580.187,A -85,B 0,C 180,E1 -30039.552,E2 -30039.552} C_VEL
LIN {X 0,Y 78.309,Z 563.756,A -85,B 0,C 180,E1 -30041.918,E2 -30041.918} C_VEL
LIN {X 0,Y 82.039,Z 548.432,A -85,B 0,C 180,E1 -30043.386,E2 -30043.386} C_VEL
LIN {X 0,Y 91.346,Z 499.133,A -85,B 0,C 180,E1 -30047.04,E2 -30047.04} C_VEL
LIN {X 0,Y 88.986,Z 489.239,A -85,B 0,C 180,E1 -30050.913,E2 -30050.913} C_VEL
LIN {X 0,Y 85.379,Z 478.525,A -85,B 0,C 180,E1 -30056.809,E2 -30056.809} C_VEL
LIN {X 0,Y 81.729,Z 468.61,A -85,B 0,C 180,E1 -30063.889,E2 -30063.889} C_VEL
LIN {X 0,Y 79.9,Z 463.593,A -85,B 0,C 180,E1 -30068.515,E2 -30068.515} C_VEL
LIN {X 0,Y 78.215,Z 459.264,A -85,B 0,C 180,E1 -30073.316,E2 -30073.316} C_VEL
LIN {X 0,Y 76.602,Z 456.193,A -85,B 0,C 180,E1 -30078.929,E2 -30078.929} C_VEL
LIN {X 0,Y 74.858,Z 452.536,A -85,B 0,C 180,E1 -30089.726,E2 -30089.726} C_VEL
LIN {X 0,Y 74.521,Z 452.459,A -85,B 0,C 180,E1 -30097.048,E2 -30097.048} C_VEL
LIN {X 0,Y 74.57,Z 452.969,A -85,B 0,C 180,E1 -30100.023,E2 -30100.023} C_VEL
LIN {X 0,Y 74.588,Z 454.262,A -85,B 0,C 180,E1 -30102.868,E2 -30102.868} C_VEL
LIN {X 0,Y 74.687,Z 457.165,A -85,B 0,C 180,E1 -30106.876,E2 -30106.876} C_VEL
LIN {X 0,Y 75.611,Z 465.486,A -85,B 0,C 180,E1 -30115.834,E2 -30115.834} C_VEL
LIN {X 0,Y 76.319,Z 467.459,A -85,B 0,C 180,E1 -30118.514,E2 -30118.514} C_VEL
LIN {X 0,Y 77.957,Z 471.097,A -85,B 0,C 180,E1 -30123.128,E2 -30123.128} C_VEL
LIN {X 0,Y 79.567,Z 475.313,A -85,B 0,C 180,E1 -30127.189,E2 -30127.189} C_VEL
LIN {X 0,Y 81.939,Z 483.387,A -85,B 0,C 180,E1 -30132.763,E2 -30132.763} C_VEL
LIN {X 0,Y 85.035,Z 493.897,A -85,B 0,C 180,E1 -30138.578,E2 -30138.578} C_VEL
LIN {X 0,Y 86.337,Z 498.328,A -85,B 0,C 180,E1 -30140.801,E2 -30140.801} C_VEL
LIN {X 0,Y 75.993,Z 549.592,A -85,B 0,C 180,E1 -30144.238,E2 -30144.238} C_VEL
LIN {X 0,Y 71.709,Z 565.33,A -85,B 0,C 180,E1 -30145.882,E2 -30145.882} C_VEL
LIN {X 0,Y 65.915,Z 581.689,A -85,B 0,C 180,E1 -30148.418,E2 -30148.418} C_VEL
LIN {X 0,Y 59.769,Z 596.092,A -85,B 0,C 180,E1 -30151.769,E2 -30151.769} C_VEL
LIN {X 0,Y 52.052,Z 611.243,A -85,B 0,C 180,E1 -30157.013,E2 -30157.013} C_VEL
LIN {X 0,Y 44.477,Z 624.728,A -85,B 0,C 180,E1 -30164.562,E2 -30164.562} C_VEL
LIN {X 0,Y 37.177,Z 637.253,A -85,B 0,C 180,E1 -30176.104,E2 -30176.104} C_VEL
LIN {X 0,Y 31.533,Z 648.372,A -85,B 0,C 180,E1 -30193.369,E2 -30193.369} C_VEL
LIN {X 0,Y 29.317,Z 656.285,A -85,B 0,C 180,E1 -30211.346,E2 -30211.346} C_VEL
LIN {X 0,Y 29.245,Z 662.563,A -85,B 0,C 180,E1 -30229.519,E2 -30229.519} C_VEL
LIN {X 0,Y 32.764,Z 669.774,A -85,B 0,C 180,E1 -30252.383,E2 -30252.383} C_VEL
LIN {X 0,Y 41.252,Z 676.629,A -85,B 0,C 180,E1 -30271.561,E2 -30271.561} C_VEL
LIN {X 0,Y 43.278,Z 677.866,A -85,B 0,C 180,E1 -30275.69,E2 -30275.69} C_VEL
LIN {X 0,Y 33.591,Z 670.976,A -85,B 0,C 180,E1 -30299.388,E2 -30299.388} C_VEL
LIN {X 0,Y 32.01,Z 667.988,A -85,B 0,C 180,E1 -30310.752,E2 -30310.752} C_VEL
LIN {X 0,Y 31.121,Z 665.159,A -85,B 0,C 180,E1 -30320.229,E2 -30320.229} C_VEL
LIN {X 0,Y 30.312,Z 658.125,A -85,B 0,C 180,E1 -30339.994,E2 -30339.994} C_VEL
LIN {X 0,Y 33.162,Z 648.072,A -85,B 0,C 180,E1 -30362.042,E2 -30362.042} C_VEL
LIN {X 0,Y 38.576,Z 637.731,A -85,B 0,C 180,E1 -30376.758,E2 -30376.758} C_VEL
LIN {X 0,Y 45.068,Z 626.423,A -85,B 0,C 180,E1 -30386.924,E2 -30386.924} C_VEL
LIN {X 0,Y 52.636,Z 613.131,A -85,B 0,C 180,E1 -30394.296,E2 -30394.296} C_VEL
LIN {X 0,Y 59.483,Z 599.581,A -85,B 0,C 180,E1 -30399.141,E2 -30399.141} C_VEL
LIN {X 0,Y 66.239,Z 584.232,A -85,B 0,C 180,E1 -30402.696,E2 -30402.696} C_VEL
LIN {X 0,Y 71.792,Z 568.584,A -85,B 0,C 180,E1 -30405.138,E2 -30405.138} C_VEL
LIN {X 0,Y 76.46,Z 551.499,A -85,B 0,C 180,E1 -30406.804,E2 -30406.804} C_VEL
LIN {X 0,Y 86.402,Z 500.754,A -85,B 0,C 180,E1 -30410.466,E2 -30410.466} C_VEL
LIN {X 0,Y 84.783,Z 493.066,A -85,B 0,C 180,E1 -30413.743,E2 -30413.743} C_VEL
LIN {X 0,Y 81.477,Z 482.553,A -85,B 0,C 180,E1 -30419.909,E2 -30419.909} C_VEL
LIN {X 0,Y 78.564,Z 473.425,A -85,B 0,C 180,E1 -30426.932,E2 -30426.932} C_VEL
LIN {X 0,Y 77.014,Z 468.822,A -85,B 0,C 180,E1 -30431.391,E2 -30431.391} C_VEL
LIN {X 0,Y 75.845,Z 465.319,A -85,B 0,C 180,E1 -30435.559,E2 -30435.559} C_VEL
LIN {X 0,Y 74.682,Z 462.763,A -85,B 0,C 180,E1 -30440.506,E2 -30440.506} C_VEL
LIN {X 0,Y 73.312,Z 459.451,A -85,B 0,C 180,E1 -30450.388,E2 -30450.388} C_VEL
LIN {X 0,Y 73.302,Z 459.574,A -85,B 0,C 180,E1 -30461.626,E2 -30461.626} C_VEL
LIN {X 0,Y 74.697,Z 463.42,A -85,B 0,C 180,E1 -30471.889,E2 -30471.889} C_VEL
LIN {X 0,Y 76.148,Z 467.035,A -85,B 0,C 180,E1 -30477.934,E2 -30477.934} C_VEL
LIN {X 0,Y 76.319,Z 467.459,A -85,B 0,C 180,E1 -30478.514,E2 -30478.514} C_VEL
LIN {X 0,Y 77.063,Z 469.529,A -85,B 0,C 180,E1 -30480.926,E2 -30480.926} C_VEL
LIN {X 0,Y 77.841,Z 473.731,A -85,B 0,C 180,E1 -30483.938,E2 -30483.938} C_VEL
LIN {X 0,Y 78.265,Z 478.643,A -85,B 0,C 180,E1 -30486.412,E2 -30486.412} C_VEL
LIN {X 0,Y 79.005,Z 489.305,A -85,B 0,C 180,E1 -30491.006,E2 -30491.006} C_VEL
LIN {X 0,Y 79.579,Z 492.635,A -85,B 0,C 180,E1 -30492.713,E2 -30492.713} C_VEL
LIN {X 0,Y 81.609,Z 500.46,A -85,B 0,C 180,E1 -30497.009,E2 -30497.009} C_VEL
LIN {X 0,Y 71.82,Z 547.315,A -85,B 0,C 180,E1 -30499.901,E2 -30499.901} C_VEL
LIN {X 0,Y 67.302,Z 563.987,A -85,B 0,C 180,E1 -30501.417,E2 -30501.417} C_VEL
LIN {X 0,Y 61.748,Z 579.524,A -85,B 0,C 180,E1 -30503.474,E2 -30503.474} C_VEL
LIN {X 0,Y 55.46,Z 593.919,A -85,B 0,C 180,E1 -30506.358,E2 -30506.358} C_VEL
LIN {X 0,Y 48.007,Z 608.308,A -85,B 0,C 180,E1 -30510.744,E2 -30510.744} C_VEL
LIN {X 0,Y 40.732,Z 620.595,A -85,B 0,C 180,E1 -30516.835,E2 -30516.835} C_VEL
LIN {X 0,Y 32.351,Z 633.721,A -85,B 0,C 180,E1 -30528.105,E2 -30528.105} C_VEL
LIN {X 0,Y 25.857,Z 644.583,A -85,B 0,C 180,E1 -30545.365,E2 -30545.365} C_VEL
LIN {X 0,Y 22.748,Z 652.947,A -85,B 0,C 180,E1 -30567.271,E2 -30567.271} C_VEL
LIN {X 0,Y 22.597,Z 659.682,A -85,B 0,C 180,E1 -30591.049,E2 -30591.049} C_VEL
LIN {X 0,Y 26.098,Z 666.223,A -85,B 0,C 180,E1 -30615.618,E2 -30615.618} C_VEL
LIN {X 0,Y 34.299,Z 672.843,A -85,B 0,C 180,E1 -30635.495,E2 -30635.495} C_VEL
LIN {X 0,Y 26.949,Z 666.989,A -85,B 0,C 180,E1 -30658.537,E2 -30658.537} C_VEL
LIN {X 0,Y 25.03,Z 663.4,A -85,B 0,C 180,E1 -30673.668,E2 -30673.668} C_VEL
LIN {X 0,Y 23.533,Z 657.504,A -85,B 0,C 180,E1 -30694.256,E2 -30694.256} C_VEL
LIN {X 0,Y 25.936,Z 647.447,A -85,B 0,C 180,E1 -30722.789,E2 -30722.789} C_VEL
LIN {X 0,Y 31.799,Z 637.169,A -85,B 0,C 180,E1 -30740.644,E2 -30740.644} C_VEL
LIN {X 0,Y 38.86,Z 625.974,A -85,B 0,C 180,E1 -30751.81,E2 -30751.81} C_VEL
LIN {X 0,Y 46.187,Z 613.958,A -85,B 0,C 180,E1 -30758.712,E2 -30758.712} C_VEL
LIN {X 0,Y 53.489,Z 600.459,A -85,B 0,C 180,E1 -30763.556,E2 -30763.556} C_VEL
LIN {X 0,Y 60.793,Z 584.785,A -85,B 0,C 180,E1 -30767.024,E2 -30767.024} C_VEL
LIN {X 0,Y 66.595,Z 569.284,A -85,B 0,C 180,E1 -30769.299,E2 -30769.299} C_VEL
LIN {X 0,Y 71.397,Z 552.82,A -85,B 0,C 180,E1 -30770.851,E2 -30770.851} C_VEL
LIN {X 0,Y 81.818,Z 502.405,A -85,B 0,C 180,E1 -30774.218,E2 -30774.218} C_VEL
LIN {X 0,Y 80.619,Z 496.662,A -85,B 0,C 180,E1 -30776.9,E2 -30776.9} C_VEL
LIN {X 0,Y 77.84,Z 486.549,A -85,B 0,C 180,E1 -30783.318,E2 -30783.318} C_VEL
LIN {X 0,Y 75.526,Z 478.245,A -85,B 0,C 180,E1 -30790.128,E2 -30790.128} C_VEL
LIN {X 0,Y 74.126,Z 473.123,A -85,B 0,C 180,E1 -30795.482,E2 -30795.482} C_VEL
LIN {X 0,Y 73.503,Z 471.181,A -85,B 0,C 180,E1 -30798.335,E2 -30798.335} C_VEL
LIN {X 0,Y 72.719,Z 469.212,A -85,B 0,C 180,E1 -30802.464,E2 -30802.464} C_VEL
LIN {X 0,Y 71.769,Z 466.383,A -85,B 0,C 180,E1 -30810.98,E2 -30810.98} C_VEL
LIN {X 0,Y 71.74,Z 466.496,A -85,B 0,C 180,E1 -30820.788,E2 -30820.788} C_VEL
LIN {X 0,Y 72.824,Z 470.097,A -85,B 0,C 180,E1 -30830.541,E2 -30830.541} C_VEL
LIN {X 0,Y 74.015,Z 473.539,A -85,B 0,C 180,E1 -30836.361,E2 -30836.361} C_VEL
LIN {X 0,Y 75.486,Z 477.484,A -85,B 0,C 180,E1 -30841.401,E2 -30841.401} C_VEL
LIN {X 0,Y 76.592,Z 480.703,A -85,B 0,C 180,E1 -30844.565,E2 -30844.565} C_VEL
LIN {X 0,Y 78.405,Z 488.008,A -85,B 0,C 180,E1 -30849.823,E2 -30849.823} C_VEL
LIN {X 0,Y 79.579,Z 492.635,A -85,B 0,C 180,E1 -30852.713,E2 -30852.713} C_VEL
LIN {X 0,Y 79.763,Z 495.469,A -85,B 0,C 180,E1 -30853.742,E2 -30853.742} C_VEL
LIN {X 0,Y 79.066,Z 499.932,A -85,B 0,C 180,E1 -30854.229,E2 -30854.229} C_VEL
LIN {X 0,Y 74.931,Z 513.4,A -85,B 0,C 180,E1 -30853.419,E2 -30853.419} C_VEL
LIN {X 0,Y 66.975,Z 549.787,A -85,B 0,C 180,E1 -30855.33,E2 -30855.33} C_VEL
LIN {X 0,Y 62.105,Z 566.482,A -85,B 0,C 180,E1 -30856.682,E2 -30856.682} C_VEL
LIN {X 0,Y 56.018,Z 582.277,A -85,B 0,C 180,E1 -30858.575,E2 -30858.575} C_VEL
LIN {X 0,Y 49.055,Z 596.86,A -85,B 0,C 180,E1 -30861.34,E2 -30861.34} C_VEL
LIN {X 0,Y 41.34,Z 610.406,A -85,B 0,C 180,E1 -30865.35,E2 -30865.35} C_VEL
LIN {X 0,Y 33.921,Z 621.973,A -85,B 0,C 180,E1 -30871.138,E2 -30871.138} C_VEL
LIN {X 0,Y 24.931,Z 634.788,A -85,B 0,C 180,E1 -30883.436,E2 -30883.436} C_VEL
LIN {X 0,Y 17.754,Z 645.959,A -85,B 0,C 180,E1 -30907.645,E2 -30907.645} C_VEL
LIN {X 0,Y 15.682,Z 652.479,A -85,B 0,C 180,E1 -30933.759,E2 -30933.759} C_VEL
LIN {X 0,Y 17.039,Z 658.978,A -85,B 0,C 180,E1 -30965.912,E2 -30965.912} C_VEL
LIN {X 0,Y 24.375,Z 666.471,A -85,B 0,C 180,E1 -30995.21,E2 -30995.21} C_VEL
LIN {X 0,Y 23.199,Z 665.589,A -85,B 0,C 180,E1 -31002.913,E2 -31002.913} C_VEL
LIN {X 0,Y 19.435,Z 661.445,A -85,B 0,C 180,E1 -31023.092,E2 -31023.092} C_VEL
LIN {X 0,Y 17.149,Z 656.776,A -85,B 0,C 180,E1 -31044.084,E2 -31044.084} C_VEL
LIN {X 0,Y 18.05,Z 648.326,A -85,B 0,C 180,E1 -31079.085,E2 -31079.085} C_VEL
LIN {X 0,Y 24.742,Z 637.226,A -85,B 0,C 180,E1 -31105.387,E2 -31105.387} C_VEL
LIN {X 0,Y 32.321,Z 626.368,A -85,B 0,C 180,E1 -31117.489,E2 -31117.489} C_VEL
LIN {X 0,Y 40.915,Z 613.327,A -85,B 0,C 180,E1 -31125.003,E2 -31125.003} C_VEL
LIN {X 0,Y 48.286,Z 600.609,A -85,B 0,C 180,E1 -31129.184,E2 -31129.184} C_VEL
LIN {X 0,Y 55.343,Z 586.264,A -85,B 0,C 180,E1 -31132.026,E2 -31132.026} C_VEL
LIN {X 0,Y 61.167,Z 571.713,A -85,B 0,C 180,E1 -31133.939,E2 -31133.939} C_VEL
LIN {X 0,Y 66.314,Z 555.316,A -85,B 0,C 180,E1 -31135.355,E2 -31135.355} C_VEL
LIN {X 0,Y 70.756,Z 535.858,A -85,B 0,C 180,E1 -31136.54,E2 -31136.54} C_VEL
LIN {X 0,Y 77.407,Z 504.227,A -85,B 0,C 180,E1 -31138.298,E2 -31138.298} C_VEL
LIN {X 0,Y 76.713,Z 500.456,A -85,B 0,C 180,E1 -31140.28,E2 -31140.28} C_VEL
LIN {X 0,Y 74.484,Z 490.664,A -85,B 0,C 180,E1 -31146.974,E2 -31146.974} C_VEL
LIN {X 0,Y 72.574,Z 482.396,A -85,B 0,C 180,E1 -31154.205,E2 -31154.205} C_VEL
LIN {X 0,Y 71.592,Z 477.808,A -85,B 0,C 180,E1 -31159.773,E2 -31159.773} C_VEL
LIN {X 0,Y 70.889,Z 475.845,A -85,B 0,C 180,E1 -31163.906,E2 -31163.906} C_VEL
LIN {X 0,Y 70.225,Z 473.29,A -85,B 0,C 180,E1 -31171.739,E2 -31171.739} C_VEL
LIN {X 0,Y 70.194,Z 473.443,A -85,B 0,C 180,E1 -31180.039,E2 -31180.039} C_VEL
LIN {X 0,Y 70.905,Z 476.545,A -85,B 0,C 180,E1 -31188.742,E2 -31188.742} C_VEL
LIN {X 0,Y 71.935,Z 480.009,A -85,B 0,C 180,E1 -31194.664,E2 -31194.664} C_VEL
LIN {X 0,Y 73.073,Z 483.791,A -85,B 0,C 180,E1 -31199.499,E2 -31199.499} C_VEL
LIN {X 0,Y 73.757,Z 486.435,A -85,B 0,C 180,E1 -31202.035,E2 -31202.035} C_VEL
LIN {X 0,Y 75.211,Z 493.132,A -85,B 0,C 180,E1 -31206.996,E2 -31206.996} C_VEL
LIN {X 0,Y 77.149,Z 502.301,A -85,B 0,C 180,E1 -31212.709,E2 -31212.709} C_VEL
LIN {X 0,Y 75.568,Z 510.445,A -85,B 0,C 180,E1 -31213.283,E2 -31213.283} C_VEL
LIN {X 0,Y 74.931,Z 513.4,A -85,B 0,C 180,E1 -31213.419,E2 -31213.419} C_VEL
LIN {X 0,Y 73.27,Z 519.085,A -85,B 0,C 180,E1 -31213.146,E2 -31213.146} C_VEL
LIN {X 0,Y 66.362,Z 537.288,A -85,B 0,C 180,E1 -31209.93,E2 -31209.93} C_VEL
LIN {X 0,Y 64.811,Z 542.982,A -85,B 0,C 180,E1 -31209.768,E2 -31209.768} C_VEL
LIN {X 0,Y 60.439,Z 559.408,A -85,B 0,C 180,E1 -31210.586,E2 -31210.586} C_VEL
LIN {X 0,Y 55.063,Z 574.555,A -85,B 0,C 180,E1 -31211.681,E2 -31211.681} C_VEL
LIN {X 0,Y 47.987,Z 590.324,A -85,B 0,C 180,E1 -31213.442,E2 -31213.442} C_VEL
LIN {X 0,Y 39.832,Z 605.088,A -85,B 0,C 180,E1 -31216.046,E2 -31216.046} C_VEL
LIN {X 0,Y 30.704,Z 619.01,A -85,B 0,C 180,E1 -31220.567,E2 -31220.567} C_VEL
LIN {X 0,Y 21.087,Z 631.638,A -85,B 0,C 180,E1 -31229.517,E2 -31229.517} C_VEL
LIN {X 0,Y 12.996,Z 641.705,A -85,B 0,C 180,E1 -31248.819,E2 -31248.819} C_VEL
LIN {X 0,Y 8.935,Z 650.614,A -85,B 0,C 180,E1 -31299.544,E2 -31299.544} C_VEL
LIN {X 0,Y 12.262,Z 657.07,A -85,B 0,C 180,E1 -31345.448,E2 -31345.448} C_VEL
LIN {X 0,Y 14.962,Z 659.452,A -85,B 0,C 180,E1 -31356.566,E2 -31356.566} C_VEL
LIN {X 0,Y 15.015,Z 659.364,A -85,B 0,C 180,E1 -31365.349,E2 -31365.349} C_VEL
LIN {X 0,Y 11.867,Z 655.877,A -85,B 0,C 180,E1 -31383.572,E2 -31383.572} C_VEL
LIN {X 0,Y 10.847,Z 647.51,A -85,B 0,C 180,E1 -31439.011,E2 -31439.011} C_VEL
LIN {X 0,Y 17.728,Z 637.536,A -85,B 0,C 180,E1 -31473.346,E2 -31473.346} C_VEL
LIN {X 0,Y 26.006,Z 627.063,A -85,B 0,C 180,E1 -31485.715,E2 -31485.715} C_VEL
LIN {X 0,Y 35.434,Z 613.854,A -85,B 0,C 180,E1 -31492.48,E2 -31492.48} C_VEL
LIN {X 0,Y 44.014,Z 599.768,A -85,B 0,C 180,E1 -31496.129,E2 -31496.129} C_VEL
LIN {X 0,Y 52.017,Z 583.983,A -85,B 0,C 180,E1 -31498.391,E2 -31498.391} C_VEL
LIN {X 0,Y 58.556,Z 567.552,A -85,B 0,C 180,E1 -31499.927,E2 -31499.927} C_VEL
LIN {X 0,Y 63.687,Z 550.562,A -85,B 0,C 180,E1 -31500.839,E2 -31500.839} C_VEL
LIN {X 0,Y 73.436,Z 505.908,A -85,B 0,C 180,E1 -31502.904,E2 -31502.904} C_VEL
LIN {X 0,Y 71.533,Z 495.986,A -85,B 0,C 180,E1 -31509.874,E2 -31509.874} C_VEL
LIN {X 0,Y 70.156,Z 487.781,A -85,B 0,C 180,E1 -31517.354,E2 -31517.354} C_VEL
LIN {X 0,Y 69.593,Z 484.023,A -85,B 0,C 180,E1 -31522.009,E2 -31522.009} C_VEL
LIN {X 0,Y 69.086,Z 482.512,A -85,B 0,C 180,E1 -31525.485,E2 -31525.485} C_VEL
LIN {X 0,Y 68.678,Z 480.34,A -85,B 0,C 180,E1 -31532.26,E2 -31532.26} C_VEL
LIN {X 0,Y 68.654,Z 480.445,A -85,B 0,C 180,E1 -31539.346,E2 -31539.346} C_VEL
LIN {X 0,Y 69.068,Z 483.078,A -85,B 0,C 180,E1 -31546.976,E2 -31546.976} C_VEL
LIN {X 0,Y 69.93,Z 486.521,A -85,B 0,C 180,E1 -31552.926,E2 -31552.926} C_VEL
LIN {X 0,Y 70.863,Z 490.663,A -85,B 0,C 180,E1 -31558.064,E2 -31558.064} C_VEL
LIN {X 0,Y 71.96,Z 497.604,A -85,B 0,C 180,E1 -31563.511,E2 -31563.511} C_VEL
LIN {X 0,Y 73.251,Z 504.608,A -85,B 0,C 180,E1 -31568.216,E2 -31568.216} C_VEL
LIN {X 0,Y 64.811,Z 542.982,A -85,B 0,C 180,E1 -31569.768,E2 -31569.768} C_VEL
LIN {X 0,Y 63.784,Z 546.785,A -85,B 0,C 180,E1 -31569.724,E2 -31569.724} C_VEL
LIN {X 0,Y 60.876,Z 554.026,A -85,B 0,C 180,E1 -31568.443,E2 -31568.443} C_VEL
LIN {X 0,Y 54.977,Z 566.238,A -85,B 0,C 180,E1 -31565.144,E2 -31565.144} C_VEL
LIN {X 0,Y 52.691,Z 571.721,A -85,B 0,C 180,E1 -31564.854,E2 -31564.854} C_VEL
LIN {X 0,Y 45.339,Z 588.44,A -85,B 0,C 180,E1 -31565.606,E2 -31565.606} C_VEL
LIN {X 0,Y 36.996,Z 603.472,A -85,B 0,C 180,E1 -31566.617,E2 -31566.617} C_VEL
LIN {X 0,Y 27.386,Z 617.662,A -85,B 0,C 180,E1 -31568.487,E2 -31568.487} C_VEL
LIN {X 0,Y 16.193,Z 631.41,A -85,B 0,C 180,E1 -31572.683,E2 -31572.683} C_VEL
LIN {X 0,Y 5.484,Z 642.689,A -85,B 0,C 180,E1 -31590.109,E2 -31590.109} C_VEL
LIN {X 0,Y 3.544,Z 649.513,A -85,B 0,C 180,E1 -31709.141,E2 -31709.141} C_VEL
LIN {X 0,Y 4.615,Z 650.557,A -85,B 0,C 180,E1 -31719.729,E2 -31719.729} C_VEL
LIN {X 0,Y 3.943,Z 649.408,A -85,B 0,C 180,E1 -31746.804,E2 -31746.804} C_VEL
LIN {X 0,Y 10.731,Z 638.438,A -85,B 0,C 180,E1 -31848.945,E2 -31848.945} C_VEL
LIN {X 0,Y 21.786,Z 626.082,A -85,B 0,C 180,E1 -31859.314,E2 -31859.314} C_VEL
LIN {X 0,Y 31.65,Z 613.084,A -85,B 0,C 180,E1 -31862.695,E2 -31862.695} C_VEL
LIN {X 0,Y 40.521,Z 598.923,A -85,B 0,C 180,E1 -31864.422,E2 -31864.422} C_VEL
LIN {X 0,Y 48.525,Z 583.381,A -85,B 0,C 180,E1 -31865.441,E2 -31865.441} C_VEL
LIN {X 0,Y 54.483,Z 568.813,A -85,B 0,C 180,E1 -31866.131,E2 -31866.131} C_VEL
LIN {X 0,Y 59.736,Z 552.352,A -85,B 0,C 180,E1 -31866.547,E2 -31866.547} C_VEL
LIN {X 0,Y 69.744,Z 508.264,A -85,B 0,C 180,E1 -31867.872,E2 -31867.872} C_VEL
LIN {X 0,Y 68.569,Z 499.798,A -85,B 0,C 180,E1 -31874.345,E2 -31874.345} C_VEL
LIN {X 0,Y 67.887,Z 492.632,A -85,B 0,C 180,E1 -31881.321,E2 -31881.321} C_VEL
LIN {X 0,Y 67.536,Z 489.736,A -85,B 0,C 180,E1 -31885.379,E2 -31885.379} C_VEL
LIN {X 0,Y 67.156,Z 487.236,A -85,B 0,C 180,E1 -31893.171,E2 -31893.171} C_VEL
LIN {X 0,Y 67.136,Z 487.375,A -85,B 0,C 180,E1 -31898.56,E2 -31898.56} C_VEL
LIN {X 0,Y 67.314,Z 489.729,A -85,B 0,C 180,E1 -31905.36,E2 -31905.36} C_VEL
LIN {X 0,Y 67.979,Z 493.283,A -85,B 0,C 180,E1 -31911.461,E2 -31911.461} C_VEL
LIN {X 0,Y 68.466,Z 496.734,A -85,B 0,C 180,E1 -31915.416,E2 -31915.416} C_VEL
LIN {X 0,Y 69.075,Z 502.932,A -85,B 0,C 180,E1 -31920.346,E2 -31920.346} C_VEL
LIN {X 0,Y 69.577,Z 506.648,A -85,B 0,C 180,E1 -31923.057,E2 -31923.057} C_VEL
LIN {X 0,Y 68.829,Z 510.415,A -85,B 0,C 180,E1 -31923.319,E2 -31923.319} C_VEL
LIN {X 0,Y 60.264,Z 547.957,A -85,B 0,C 180,E1 -31924.185,E2 -31924.185} C_VEL
LIN {X 0,Y 55.429,Z 564.246,A -85,B 0,C 180,E1 -31924.613,E2 -31924.613} C_VEL
LIN {X 0,Y 52.691,Z 571.721,A -85,B 0,C 180,E1 -31924.854,E2 -31924.854} C_VEL
LIN {X 0,Y 50.315,Z 577.105,A -85,B 0,C 180,E1 -31924.508,E2 -31924.508} C_VEL
LIN {X 0,Y 45.408,Z 585.359,A -85,B 0,C 180,E1 -31921.555,E2 -31921.555} C_VEL
LIN {X 0,Y 40.163,Z 593.372,A -85,B 0,C 180,E1 -31917.642,E2 -31917.642} C_VEL
LIN {X 0,Y 37.082,Z 598.401,A -85,B 0,C 180,E1 -31916.333,E2 -31916.333} C_VEL
LIN {X 0,Y 28,Z 612.729,A -85,B 0,C 180,E1 -31914.669,E2 -31914.669} C_VEL
LIN {X 0,Y 18.231,Z 625.699,A -85,B 0,C 180,E1 -31910.455,E2 -31910.455} C_VEL
LIN {X 0,Y 8.47,Z 637.104,A -85,B 0,C 180,E1 -31894.052,E2 -31894.052} C_VEL
LIN {X 0,Y 8.156,Z 637.495,A -85,B 0,C 180,E1 -31890.636,E2 -31890.636} C_VEL
LIN {X 0,Y 18.932,Z 625.39,A -85,B 0,C 180,E1 -31877.887,E2 -31877.887} C_VEL
LIN {X 0,Y 29.103,Z 611.994,A -85,B 0,C 180,E1 -31875.078,E2 -31875.078} C_VEL
LIN {X 0,Y 38.016,Z 597.898,A -85,B 0,C 180,E1 -31874.006,E2 -31874.006} C_VEL
LIN {X 0,Y 46.05,Z 582.404,A -85,B 0,C 180,E1 -31873.422,E2 -31873.422} C_VEL
LIN {X 0,Y 51.874,Z 568.121,A -85,B 0,C 180,E1 -31873.203,E2 -31873.203} C_VEL
LIN {X 0,Y 56.791,Z 552.764,A -85,B 0,C 180,E1 -31873.003,E2 -31873.003} C_VEL
LIN {X 0,Y 62.002,Z 530.66,A -85,B 0,C 180,E1 -31873.105,E2 -31873.105} C_VEL
LIN {X 0,Y 66.527,Z 510.533,A -85,B 0,C 180,E1 -31873.35,E2 -31873.35} C_VEL
LIN {X 0,Y 66.026,Z 502.772,A -85,B 0,C 180,E1 -31879.972,E2 -31879.972} C_VEL
LIN {X 0,Y 65.792,Z 497.191,A -85,B 0,C 180,E1 -31885.967,E2 -31885.967} C_VEL
LIN {X 0,Y 65.722,Z 495.886,A -85,B 0,C 180,E1 -31888.18,E2 -31888.18} C_VEL
LIN {X 0,Y 65.639,Z 494.156,A -85,B 0,C 180,E1 -31894.041,E2 -31894.041} C_VEL
LIN {X 0,Y 65.615,Z 494.355,A -85,B 0,C 180,E1 -31897.889,E2 -31897.889} C_VEL
LIN {X 0,Y 65.608,Z 496.342,A -85,B 0,C 180,E1 -31903.595,E2 -31903.595} C_VEL
LIN {X 0,Y 65.979,Z 499.861,A -85,B 0,C 180,E1 -31909.527,E2 -31909.527} C_VEL
LIN {X 0,Y 66.236,Z 503.409,A -85,B 0,C 180,E1 -31913.113,E2 -31913.113} C_VEL
LIN {X 0,Y 66.499,Z 509.209,A -85,B 0,C 180,E1 -31917.706,E2 -31917.706} C_VEL
LIN {X 0,Y 57.668,Z 547.646,A -85,B 0,C 180,E1 -31917.743,E2 -31917.743} C_VEL
LIN {X 0,Y 52.92,Z 563.737,A -85,B 0,C 180,E1 -31917.606,E2 -31917.606} C_VEL
LIN {X 0,Y 47.002,Z 578.814,A -85,B 0,C 180,E1 -31917.259,E2 -31917.259} C_VEL
LIN {X 0,Y 40.026,Z 593.148,A -85,B 0,C 180,E1 -31916.738,E2 -31916.738} C_VEL
LIN {X 0,Y 37.082,Z 598.401,A -85,B 0,C 180,E1 -31916.333,E2 -31916.333} C_VEL
LIN {X 0,Y 34.969,Z 601.646,A -85,B 0,C 180,E1 -31914.914,E2 -31914.914} C_VEL
LIN {X 0,Y 31.374,Z 606.295,A -85,B 0,C 180,E1 -31909.198,E2 -31909.198} C_VEL
LIN {X 0,Y 28.07,Z 610.847,A -85,B 0,C 180,E1 -31901.922,E2 -31901.922} C_VEL
LIN {X 0,Y 26.011,Z 613.946,A -85,B 0,C 180,E1 -31898.819,E2 -31898.819} C_VEL
LIN {X 0,Y 23.73,Z 617.37,A -85,B 0,C 180,E1 -31896.328,E2 -31896.328} C_VEL
LIN {X 0,Y 24.833,Z 615.832,A -85,B 0,C 180,E1 -31891.941,E2 -31891.941} C_VEL
LIN {X 0,Y 33.235,Z 602.708,A -85,B 0,C 180,E1 -31886.053,E2 -31886.053} C_VEL
LIN {X 0,Y 41.042,Z 588.315,A -85,B 0,C 180,E1 -31883.052,E2 -31883.052} C_VEL
LIN {X 0,Y 47.588,Z 573.686,A -85,B 0,C 180,E1 -31881.246,E2 -31881.246} C_VEL
LIN {X 0,Y 53.357,Z 557.09,A -85,B 0,C 180,E1 -31880.238,E2 -31880.238} C_VEL
LIN {X 0,Y 57.581,Z 540.893,A -85,B 0,C 180,E1 -31879.624,E2 -31879.624} C_VEL
LIN {X 0,Y 63.955,Z 512.814,A -85,B 0,C 180,E1 -31879.399,E2 -31879.399} C_VEL
LIN {X 0,Y 63.923,Z 505.207,A -85,B 0,C 180,E1 -31886.644,E2 -31886.644} C_VEL
LIN {X 0,Y 64.072,Z 502.547,A -85,B 0,C 180,E1 -31889.898,E2 -31889.898} C_VEL
LIN {X 0,Y 64.133,Z 501.086,A -85,B 0,C 180,E1 -31894.765,E2 -31894.765} C_VEL
LIN {X 0,Y 64.103,Z 501.323,A -85,B 0,C 180,E1 -31897.198,E2 -31897.198} C_VEL
LIN {X 0,Y 63.962,Z 503.014,A -85,B 0,C 180,E1 -31901.834,E2 -31901.834} C_VEL
LIN {X 0,Y 64.009,Z 506.065,A -85,B 0,C 180,E1 -31906.809,E2 -31906.809} C_VEL
LIN {X 0,Y 63.974,Z 510.774,A -85,B 0,C 180,E1 -31911.078,E2 -31911.078} C_VEL
LIN {X 0,Y 63.973,Z 511.415,A -85,B 0,C 180,E1 -31911.576,E2 -31911.576} C_VEL
LIN {X 0,Y 56.686,Z 543.35,A -85,B 0,C 180,E1 -31911.027,E2 -31911.027} C_VEL
LIN {X 0,Y 52,Z 560.369,A -85,B 0,C 180,E1 -31910.239,E2 -31910.239} C_VEL
LIN {X 0,Y 46.533,Z 575.351,A -85,B 0,C 180,E1 -31909.044,E2 -31909.044} C_VEL
LIN {X 0,Y 39.378,Z 590.966,A -85,B 0,C 180,E1 -31906.895,E2 -31906.895} C_VEL
LIN {X 0,Y 31.063,Z 605.905,A -85,B 0,C 180,E1 -31902.75,E2 -31902.75} C_VEL
LIN {X 0,Y 26.011,Z 613.946,A -85,B 0,C 180,E1 -31898.819,E2 -31898.819} C_VEL
LIN {X 0,Y 26.389,Z 613.313,A -85,B 0,C 180,E1 -31896.729,E2 -31896.729} C_VEL
LIN {X 0,Y 27.022,Z 612.312,A -85,B 0,C 180,E1 -31895.656,E2 -31895.656} C_VEL
LIN {X 0,Y 31.053,Z 605.7,A -85,B 0,C 180,E1 -31893.65,E2 -31893.65} C_VEL
LIN {X 0,Y 36.659,Z 595.454,A -85,B 0,C 180,E1 -31893.341,E2 -31893.341} C_VEL
LIN {X 0,Y 39.667,Z 589.32,A -85,B 0,C 180,E1 -31892.859,E2 -31892.859} C_VEL
LIN {X 0,Y 42.483,Z 583.087,A -85,B 0,C 180,E1 -31891.767,E2 -31891.767} C_VEL
LIN {X 0,Y 48.265,Z 568.571,A -85,B 0,C 180,E1 -31889.138,E2 -31889.138} C_VEL
LIN {X 0,Y 53.202,Z 552.871,A -85,B 0,C 180,E1 -31887.459,E2 -31887.459} C_VEL
LIN {X 0,Y 58.339,Z 531.02,A -85,B 0,C 180,E1 -31886.231,E2 -31886.231} C_VEL
LIN {X 0,Y 61.86,Z 515.371,A -85,B 0,C 180,E1 -31885.727,E2 -31885.727} C_VEL
LIN {X 0,Y 62.487,Z 509.001,A -85,B 0,C 180,E1 -31892.429,E2 -31892.429} C_VEL
LIN {X 0,Y 62.626,Z 508.084,A -85,B 0,C 180,E1 -31895.728,E2 -31895.728} C_VEL
LIN {X 0,Y 62.376,Z 509.756,A -85,B 0,C 180,E1 -31900.179,E2 -31900.179} C_VEL
LIN {X 0,Y 62.203,Z 511.995,A -85,B 0,C 180,E1 -31903.566,E2 -31903.566} C_VEL
LIN {X 0,Y 62.056,Z 513.704,A -85,B 0,C 180,E1 -31905.178,E2 -31905.178} C_VEL
LIN {X 0,Y 55.776,Z 541.662,A -85,B 0,C 180,E1 -31903.965,E2 -31903.965} C_VEL
LIN {X 0,Y 51.292,Z 558.993,A -85,B 0,C 180,E1 -31902.539,E2 -31902.539} C_VEL
LIN {X 0,Y 46.174,Z 573.937,A -85,B 0,C 180,E1 -31900.465,E2 -31900.465} C_VEL
LIN {X 0,Y 39.522,Z 589.551,A -85,B 0,C 180,E1 -31896.772,E2 -31896.772} C_VEL
LIN {X 0,Y 38.557,Z 591.514,A -85,B 0,C 180,E1 -31896.101,E2 -31896.101} C_VEL
LIN {X 0,Y 38.633,Z 591.379,A -85,B 0,C 180,E1 -31894.096,E2 -31894.096} C_VEL
LIN {X 0,Y 42.483,Z 583.087,A -85,B 0,C 180,E1 -31891.767,E2 -31891.767} C_VEL
LIN {X 0,Y 45.512,Z 575.75,A -85,B 0,C 180,E1 -31891.121,E2 -31891.121} C_VEL
LIN {X 0,Y 48.185,Z 568.26,A -85,B 0,C 180,E1 -31891.858,E2 -31891.858} C_VEL
LIN {X 0,Y 52.683,Z 553.054,A -85,B 0,C 180,E1 -31894.077,E2 -31894.077} C_VEL
LIN {X 0,Y 54.583,Z 545.156,A -85,B 0,C 180,E1 -31894.261,E2 -31894.261} C_VEL
LIN {X 0,Y 55.165,Z 542.521,A -85,B 0,C 180,E1 -31894.025,E2 -31894.025} C_VEL
LIN {X 0,Y 60.528,Z 518.034,A -85,B 0,C 180,E1 -31892.544,E2 -31892.544} C_VEL
LIN {X 0,Y 61.004,Z 515.571,A -85,B 0,C 180,E1 -31895.174,E2 -31895.174} C_VEL
LIN {X 0,Y 60.999,Z 515.694,A -85,B 0,C 180,E1 -31896.704,E2 -31896.704} C_VEL
LIN {X 0,Y 60.826,Z 516.575,A -85,B 0,C 180,E1 -31898.334,E2 -31898.334} C_VEL
LIN {X 0,Y 58.979,Z 525.053,A -85,B 0,C 180,E1 -31897.98,E2 -31897.98} C_VEL
LIN {X 0,Y 52.765,Z 552.728,A -85,B 0,C 180,E1 -31895.405,E2 -31895.405} C_VEL
LIN {X 0,Y 52.736,Z 552.829,A -85,B 0,C 180,E1 -31895.178,E2 -31895.178} C_VEL
LIN {X 0,Y 55.165,Z 542.521,A -85,B 0,C 180,E1 -31894.025,E2 -31894.025} C_VEL
LIN {X 0,Y 58.689,Z 543,A -85,B 0,C 180,E1 -31892.247,E2 -31892.247} C_VEL
LIN {X 0,Y 58.689,Z 600,A -85,B 0,C 180,E1 -31892.247,E2 -31892.247} C_VEL
LIN {X 0,Y 58.689,Z 600,A -85,B 0,C 180,E1 -31892.247,E2 -31892.247}

QRS_NEXT_CUT()

QRS_NEXT()
QRS_HOME()

END
